Universal Robots URScript: Test Teach Position.script

def Test_Teach_Position():
  global _hidden_verificationVariable=0
  set_tcp(p[-4.516483728619642E-6,-4.494070941040221E-6,-3.385497268221845E-5,0.0,0.0,0.0])
  set_safety_mode_transition_hardness(1)
  set_tool_communication(False, 115200, 0, 1, 1.5, 3.5)
  set_tool_output_mode(0)
  set_tool_digital_output_mode(0, 1)
  set_tool_digital_output_mode(1, 1)
  set_tool_voltage(0)
  set_target_payload(0.000000, [0.000000, 0.000000, 0.000000], [0.000000, 0.000000, 0.000000, 0.000000, 0.000000, 0.000000])
  set_standard_analog_input_domain(0, 1)
  set_standard_analog_input_domain(1, 1)
  set_tool_analog_input_domain(0, 1)
  set_tool_analog_input_domain(1, 1)
  set_analog_outputdomain(0, 0)
  set_analog_outputdomain(1, 0)
  set_input_actions_to_default()
  set_gravity([0.0, 0.0, 9.82])
  global Point_1=p[0.0,0.0,0.0,0.0,0.0,0.0]
  # begin: URCap Installation Node
  #   Source: MachineLogic for Universal Robots, 3.1.7, Vention Inc.
  #   Type: MachineLogic for Universal Robots
  def waitForResponse(expected_response_vention, cname_vention):
  response_vention = socket_read_string(cname_vention,timeout=15)
  while response_vention != expected_response_vention:
  sleep(0.01)
  response_vention = socket_read_string(cname_vention,timeout=15)
  end
  sleep(0.01)
  sync()
  end
  def sendString(string_vention, expected_response_vention, cname_vention):
  socket_send_string(str_cat(string_vention,";"), cname_vention)
  response_vention = socket_read_string(cname_vention,timeout=15)
  if(response_vention == "nAck"):
  popup("nAck received")
  end
  while response_vention != expected_response_vention:
  sleep(0.01)
  response_vention = socket_read_string(cname_vention,timeout=15)
  if(response_vention == "nAck"):
  popup("nAck received")
  end
  end
  sleep(0.01)
  sync()
  end
  def sendStringNAck(string_vention, expected_response_vention, cname_vention):
  socket_send_string(str_cat(string_vention,";"), cname_vention)
  response_vention = socket_read_string(cname_vention,timeout=15)
  if(response_vention == "nAck"):
  popup("nAck received")
  end
  while(response_vention != expected_response_vention and response_vention != "nAck"):
  sleep(0.01)
  response_vention = socket_read_string(cname_vention,timeout=15)
  if(response_vention == "nAck"):
  popup("nAck received",blocking=True)
  end
  end
  sleep(0.01)
  sync()
  end
  def sendStringWithTimeout(string_vention, expected_response_vention, cname_vention):
  socket_send_string(str_cat(string_vention,";"), cname_vention)
  response_vention = socket_read_string(cname_vention,timeout=10)
  if(response_vention == "nAck"):
  popup("nAck received"+string_vention)
  end
  sleep(0.01)
  sync()
  end
  def pollString(string_vention, expected_response_vention, cname_vention):
  socket_send_string(str_cat(string_vention,";"), cname_vention)
  response_vention = socket_read_string(cname_vention,timeout=15)
  if(response_vention == "nAck"):
  popup("nAck received")
  end
  while response_vention != expected_response_vention:
  sleep(1)
  socket_send_string(str_cat(string_vention,";"), cname_vention)
  response_vention = socket_read_string(cname_vention,timeout=15)
  if(response_vention == "nAck"):
  popup("nAck received")
  end
  end
  sleep(0.01)
  sync()
  end
  def sendVariable(var_vention, data_vention, expected_response_vention, cname_vention):
  socket_set_var(var_vention, data_vention, cname_vention)
  response_vention = socket_read_string(cname_vention,timeout=15)
  if(response_vention == "nAck"):
  popup("nAck received")
  end
  while response_vention != expected_response_vention:
  sleep(0.01)
  response_vention = socket_read_string(cname_vention,timeout=15)
  if(response_vention == "nAck"):
  popup("nAck received")
  end
  end
  sleep(0.01)
  sync()
  end
  def intToString(integer_vention,cname_vention):
  stringFix=""
  multiplier_vention123=1
  if integer_vention<0:
  stringFix="-"
  multiplier_vention123=-1
  end
  socket_set_var("GetString",integer_vention*multiplier_vention123,cname_vention)
  string_vention=""
  while string_vention=="":
  sleep(0.01)
  string_vention=socket_read_string(cname_vention,timeout=15)
  end
  sleep(0.01)
  sync()
  string_vention=stringFix+string_vention
  return string_vention
  end
  string_vention=""
  isVentionMovementBusy = False
  isVentionParallelMovementSendingScript = False
  ventionThreadHandle = 1
  isVentionMovementBusyMachineMotion1 = False
  isVentionParallelMovementSendingScriptMachineMotion1 = False
  socket_vention = socket_open("192.168.3.52", 9999, "MachineMotion1")
  if socket_vention==False:
  popup("Check configuration, can't connect to MachineMotion")
  end
  waitForResponse("MachineMotion connection established", "MachineMotion1")
  sendString("isReady", "MachineMotion isReady = true", "MachineMotion1")
  sendStringWithTimeout("setURCapVersion2", "setURCapVersion loaded", "MachineMotion1")
  sendString("SET speed_v2 1000000", "Ack", "MachineMotion1")
  sendString("SET acceleration_v2 100000", "Ack", "MachineMotion1")
  sendString("SET de_axis_1_microsteps_config 8", "Ack", "MachineMotion1")
  sendString("SET de_axis_1_mechanical_gain_config_v2 150000.0", "Ack", "MachineMotion1")
  sendString("SET de_axis_1_direction_config 1", "Ack", "MachineMotion1")
  sendString("SET de_axis_1_type_config Custom Actuator ", "Ack", "MachineMotion1")
  sendString("de_axis_1_config_exec", "Ack", "MachineMotion1")
  # end: URCap Installation Node
  step_count_8ae00f07_a168_4cef_8ff5_9bbe05fd2c44 = 0.0
  thread Step_Counter_Thread_d5810124_ed15_46ca_96ea_71c010d4b624():
    while (True):
      step_count_8ae00f07_a168_4cef_8ff5_9bbe05fd2c44 = step_count_8ae00f07_a168_4cef_8ff5_9bbe05fd2c44 + 1.0
      sync()
    end
  end
  run Step_Counter_Thread_d5810124_ed15_46ca_96ea_71c010d4b624()
  global freedrive_m_var=  False
  global Waypoint_1_p=p[.574920139234, .290181243295, .475641456904, -.083548844531, 2.369773198085, -.198339248333]
  global Waypoint_1_q=[0.947482705116272, -1.4870131772807618, -2.5590596199035645, -0.2591535610011597, 0.8874344825744629, 2.3016035556793213]
  $ 17 "Thread_1"
  thread Thread_1():
    while (True):
      $ 18 "Loop  True "
      while (  True  ):
        $ 19 "If freedrive_m_var≟ True "
        if (freedrive_m_var ==   True  ):
          $ 20 "freedrive_mode()"
          freedrive_mode()
        else:
          $ 21 "Else" "noBreak"
          $ 22 "end_freedrive_mode()"
          end_freedrive_mode()
        end
        $ 23 "sync()"
        sync()
      end
    end
  end
  threadId_Thread_1 = run Thread_1()
  $ 2 "Robot Program"
  $ 3 "Home"
  movej([-1.5370344946663685, -1.5288164776614686, -2.7875118543223336, -0.3724559904209972, 1.623548359823722, -0.03990680376161748], a=1.3962634015954636, v=1.0471975511965976)
  $ 4 "MoveJ"
  $ 5 "Waypoint_1" "breakAfter"
  movej(get_inverse_kin(Waypoint_1_p, qnear=Waypoint_1_q), a=1.3962634015954636, v=1.0471975511965976)
  $ 6 "freedrive_m_var≔ False "
  global freedrive_m_var=  False
  $ 7 "freedrive_m_var≔ True "
  global freedrive_m_var=  True
  $ 8 "Popup: Move the robot to the peg center, then click OK"
  popup("Move the robot to the peg center, then click OK", "Message", False, False, blocking=True)
  $ 9 "freedrive_m_var≔ False "
  global freedrive_m_var=  False
  $ 10 "Wait: 0.25"
  sleep(0.25)
  $ 11 "sync()"
  sync()
  $ 12 "tcp_pose≔get_actual_tcp_pose()"
  global tcp_pose= get_actual_tcp_pose ()
  $ 13 "Home"
  movej([-1.5370344946663685, -1.5288164776614686, -2.7875118543223336, -0.3724559904209972, 1.623548359823722, -0.03990680376161748], a=1.3962634015954636, v=1.0471975511965976)
  $ 14 "MoveJ"
  $ 15 "tcp_pose" "breakAfter"
  movej(tcp_pose, a=1.3962634015954636, v=1.0471975511965976)
  $ 16 "Home"
  movej([-1.5370344946663685, -1.5288164776614686, -2.7875118543223336, -0.3724559904209972, 1.623548359823722, -0.03990680376161748], a=1.3962634015954636, v=1.0471975511965976)
end
